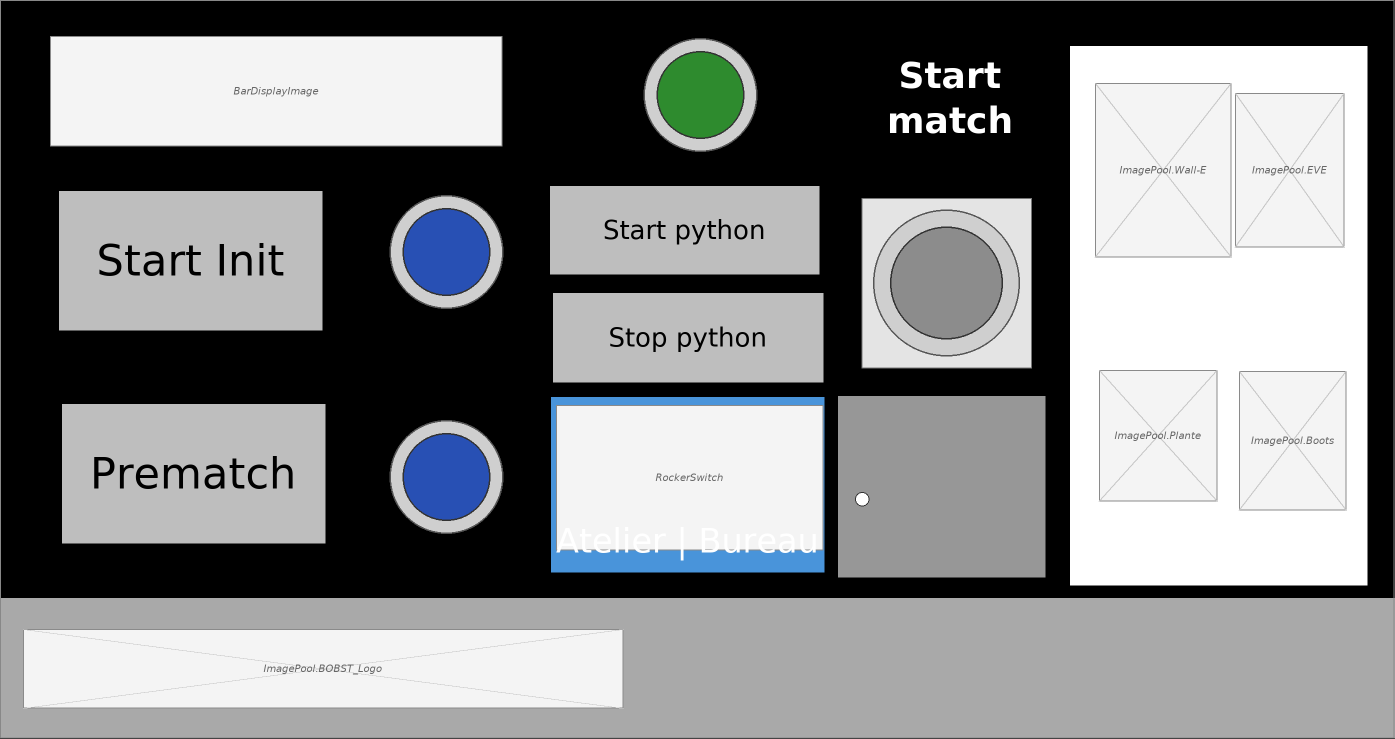
VISUALIZATION V_Init  // 1395x739
    Rectangle (-1,598 1396x140)
    RoundedRectangle (550,396 275x177)
    RoundedRectangle (1069,45 299x541)
    RoundedRectangle (837,395 209x183)
    Lamp1 (374,186 145x132), variable: G_init.ietapeInit <> 0, style: Lamp-Lamp1-Blue
    RockerSwitch (556,405 267x145), variable: G_Visus.bInitChoixCote, behaviour: TOGGLE, style: Switch-RockerSwitch-Gray
    BarDisplayImage (50,36 452x110), value: G_Visus.iInitProgressBar, style: BarDisplayImage-Gray, scale format: %.1f, scale 0..100
    Lamp1 (374,411 145x132), variable: G_PreMatch.bPrematchActive, style: Lamp-Lamp1-Blue
    Label (519,501 337x79), "Atelier | Bureau"
    RoundedRectangle (58,190 265x141), "Start Init"
        OnMouseDown: toggle G_Visus.bInitStart
        OnMouseUp: toggle G_Visus.bInitStart
    RoundedRectangle (61,403 265x141), "Prematch"
        OnMouseDown: toggle G_Visus.bInitPrematch
        OnMouseUp: toggle G_Visus.bInitPrematch
    RadioButton (853,434 178x130), variable: G_Visus.iInitChoixParcours
        Areas[0]: Text=Radiobutton
        Areas[1]: Text=Radiobutton
        p340057476: Parcours 1
        p3123465237: Parcours 2
        p2481256679: Parcours 3
    RoundedRectangle (1185,980 0x2)
    Image (1095,83 136x174), image: ImagePool.Wall-E
    Image (1235,93 109x154), image: ImagePool.EVE
    Image (1099,370 118x131), image: ImagePool.Plante
    Image (1239,371 107x139), image: ImagePool.Boots
    Lamp1 (628,29 145x132), variable: G_Visus.bInitPyScriptRunning, style: Lamp-Lamp1-Green
    RoundedRectangle (549,185 271x90), "Start python"
        OnMouseDown: toggle G_Visus.bInitStartPyscript
        OnMouseUp: toggle G_Visus.bInitStartPyscript
    RoundedRectangle (552,292 272x91), "Stop python"
        OnMouseDown: toggle G_Visus.bInitStopPyscript
        OnMouseUp: toggle G_Visus.bInitStopPyscript
    PushSwitch (849,198 195x170), variable: G_Visus.bInitStartMatch, behaviour: TAP, style: Switch-PushSwitch-Gray
    Label (857,46 186x104), "Start match"
    Image (23,629 600x79), image: ImagePool.BOBST_Logo
        OnMouseDown: change screen: V_Menu
END_VISUALIZATION

(* stored: Version 1.1.0.1, ProductVersion 3.1.4024.12
   Visu V_Init: Id {7b75c880-1704-4f3c-9bad-4d11c105fb89} *)
